Yaskawa INFORM job: AAA.JBI

/JOB
//NAME AAA
//POS
///NPOS 51,0,0,0,0,0
///TOOL 10
///POSTYPE PULSE
///PULSE
C00000=-69499,-30257,-42570,-18909,-69402,74527
C00001=-69549,-32276,-45094,-20883,-70341,73613
C00002=-68847,-33623,-46778,-21857,-71568,72091
C00003=-68061,-34801,-48261,-22885,-72842,70541
C00004=-67255,-35930,-49660,-24059,-74096,69042
C00005=-66373,-36997,-50948,-25288,-75318,67573
C00006=-65393,-38019,-52126,-26535,-76486,66139
C00007=-64319,-39049,-53236,-27798,-77570,64761
C00008=-63152,-40136,-54305,-29073,-78541,63450
C00009=-61875,-41281,-55326,-30328,-79393,62200
C00010=-60465,-42441,-56253,-31523,-80139,60996
C00011=-58901,-43548,-57035,-32621,-80798,59821
C00012=-57177,-44547,-57634,-33605,-81387,58667
C00013=-55295,-45402,-58034,-34469,-81917,57533
C00014=-53265,-46094,-58229,-35219,-82391,56420
C00015=-51099,-46612,-58224,-35858,-82815,55330
C00016=-48805,-46947,-58019,-36390,-83192,54265
C00017=-46393,-47090,-57619,-36817,-83528,53227
C00018=-43871,-47043,-57031,-37139,-83826,52216
C00019=-41248,-46811,-56265,-37358,-84088,51235
C00020=-38527,-46401,-55330,-37470,-84316,50284
C00021=-35710,-45808,-54226,-37469,-84518,49362
C00022=-32796,-45014,-52944,-37344,-84709,48466
C00023=-29780,-43989,-51469,-37080,-84908,47593
C00024=-26661,-42711,-49788,-36668,-85136,46741
C00025=-23433,-41173,-47899,-36096,-85405,45907
C00026=-20094,-39388,-45815,-35355,-85721,45093
C00027=-16638,-37379,-43552,-34434,-86086,44298
C00028=-13056,-35157,-41123,-33319,-86506,43524
C00029=-9338,-32714,-38530,-31995,-86998,42766
C00030=-5474,-30023,-35771,-30448,-87587,42021
C00031=-1462,-27060,-32849,-28674,-88300,41285
C00032=2698,-23819,-29786,-26676,-89155,40557
C00033=6992,-20316,-26627,-24470,-90160,39837
C00034=11396,-16568,-23425,-22087,-91317,39126
C00035=15870,-12581,-20228,-19576,-92632,38422
C00036=20359,-8345,-17076,-17003,-94115,37720
C00037=24796,-3848,-14001,-14451,-95774,37014
C00038=29106,930,-11018,-12009,-97612,36294
C00039=33215,6015,-8121,-9767,-99636,35548
C00040=37059,11434,-5295,-7809,-101849,34761
C00041=40585,17162,-2543,-6201,-104228,33920
C00042=43770,23088,82,-4980,-106701,33021
C00043=46614,29074,2518,-4155,-109182,32065
C00044=49128,35070,4755,-3731,-111637,31047
C00045=51316,41089,6814,-3723,-114072,29952
C00046=53199,47042,8657,-4132,-116433,28776
C00047=54816,52823,10233,-4927,-118655,27526
C00048=56204,58383,11523,-6075,-120706,26208
C00049=57447,63448,12428,-7454,-122415,24887
C00050=58534,68041,12995,-9088,-123781,23559
//INST
///DATE 2023/03/24 18:38
///ATTR SC,RW
///GROUP1 RB1
NOP
MOVJ C00000 VJ=50.0
MOVL C00001 V=50.0
MOVL C00002 V=50.0
MOVL C00003 V=50.0
MOVL C00004 V=50.0
MOVL C00005 V=50.0
MOVL C00006 V=50.0
MOVL C00007 V=50.0
MOVL C00008 V=50.0
MOVL C00009 V=50.0
MOVL C00010 V=50.0
MOVL C00011 V=50.0
MOVL C00012 V=50.0
MOVL C00013 V=50.0
MOVL C00014 V=50.0
MOVL C00015 V=50.0
MOVL C00016 V=50.0
MOVL C00017 V=50.0
MOVL C00018 V=50.0
MOVL C00019 V=50.0
MOVL C00020 V=50.0
MOVL C00021 V=50.0
MOVL C00022 V=50.0
MOVL C00023 V=50.0
MOVL C00024 V=50.0
MOVL C00025 V=50.0
MOVL C00026 V=50.0
MOVL C00027 V=50.0
MOVL C00028 V=50.0
MOVL C00029 V=50.0
MOVL C00030 V=50.0
MOVL C00031 V=50.0
MOVL C00032 V=50.0
MOVL C00033 V=50.0
MOVL C00034 V=50.0
MOVL C00035 V=50.0
MOVL C00036 V=50.0
MOVL C00037 V=50.0
MOVL C00038 V=50.0
MOVL C00039 V=50.0
MOVL C00040 V=50.0
MOVL C00041 V=50.0
MOVL C00042 V=50.0
MOVL C00043 V=50.0
MOVL C00044 V=50.0
MOVL C00045 V=50.0
MOVL C00046 V=50.0
MOVL C00047 V=50.0
MOVL C00048 V=50.0
MOVL C00049 V=50.0
MOVL C00050 V=50.0
END
